(* IEC 61131-3 sources: AXOpen/src/components.abstractions/ctrl/src/AxoDrives (part 2) *)

(* ---- AxoDrive.st ---- *)
USING AXOpen.Core;
USING AXOpen.Messaging.Static;
USING AXOpen.Messaging;
USING System.Strings;

NAMESPACE AXOpen.Components.Abstractions.AxoDrives
    {#ix-attr:[Container(Layout.Wrap)]}
    CLASS PUBLIC ABSTRACT AxoDrive EXTENDS AXOpen.Core.AxoComponent IMPLEMENTS AXOpen.Components.Abstractions.AxoDrives.IAxoDrive
        VAR PUBLIC
            {#ix-attr:[Container(Layout.Wrap)]}
            {#ix-attr:[ComponentHeader()]}
            {#ix-attr:[ReadOnly()]}
            {#ix-set:AttributeName = "<#Drive state#>"}
            DriveState          :   AXOpen.Components.Abstractions.AxoDrives.eAxoDriveState;

            DriveStatus         :   AxoDrive_Status;
            Messenger           :   AXOpen.Messaging.Static.AxoMessenger;
            TaskMessenger       :   AXOpen.Messaging.Static.AxoMessenger;
        END_VAR

        VAR PUBLIC
            {#ix-attr:[Container(Layout.Wrap)]}
            {#ix-attr:[ComponentDetails("Tasks")]}
            {#ix-set:AttributeName = "<#Restore#>"}
            RestoreTask : AXOpen.Core.AxoTask;
            //***********Power********************************
            {#ix-attr:[Container(Layout.UniformGrid)]}
            {#ix-attr:[Group(GroupLayout.GroupBox)]}
            {#ix-attr:[ComponentDetails("Tasks")]}
            {#ix-set:AttributeName = "<#Power task#>"}
            AxoPower_Task                           :   AXOpen.Components.Abstractions.AxoDrives.Axo_Power;
            {#ix-attr:[ComponentDetails("Tasks")]}
            {#ix-set:AttributeName = "<#Power status#>"}
            AxoPower_Status                         :   BOOL;
            {#ix-attr:[ComponentDetails("Tasks")]}
            {#ix-set:AttributeName = "<#Power valid#>"}
            AxoPower_Valid                          :   BOOL;
            {#ix-attr:[ComponentDetails("Tasks")]}
            {#ix-set:AttributeName = "<#Power error#>"}
            AxoPower_Error                          :   BOOL;
            {#ix-attr:[ComponentDetails("Tasks")]}
            {#ix-set:AttributeName = "<#Power error ID#>"}
            AxoPower_ErrorID                        :   WORD;
            //***********Stop*********************************
            {#ix-attr:[Container(Layout.UniformGrid)]}
            {#ix-attr:[Group(GroupLayout.GroupBox)]}
            {#ix-attr:[ComponentDetails("Tasks")]}
            {#ix-set:AttributeName = "<#Stop task#>"}
            AxoStop_Task                            :   AXOpen.Core.AxoTask;
            {#ix-attr:[ComponentDetails("Tasks")]}
            {#ix-set:AttributeName = "<#Stop decceleration#>"}
            AxoStop_Deceleration                    :   LREAL;
            {#ix-attr:[ComponentDetails("Tasks")]}
            {#ix-set:AttributeName = "<#Stop jerk#>"}
            AxoStop_Jerk                            :   LREAL;
            {#ix-attr:[ComponentDetails("Tasks")]}
            {#ix-set:AttributeName = "<#Stop done#>"}
            AxoStop_Done                            :   BOOL;
            {#ix-attr:[ComponentDetails("Tasks")]}
            {#ix-set:AttributeName = "<#Stop busy#>"}
            AxoStop_Busy                            :   BOOL;
            {#ix-attr:[ComponentDetails("Tasks")]}
            {#ix-set:AttributeName = "<#Stop active#>"}
            AxoStop_Active                          :   BOOL;
            {#ix-attr:[ComponentDetails("Tasks")]}
            {#ix-set:AttributeName = "<#Stop aborted#>"}
            AxoStop_CommandAborted                  :   BOOL;
            {#ix-attr:[ComponentDetails("Tasks")]}
            {#ix-set:AttributeName = "<#Stop error#>"}
            AxoStop_Error                           :   BOOL;
            {#ix-attr:[ComponentDetails("Tasks")]}
            {#ix-set:AttributeName = "<#Stop error ID#>"}
            AxoStop_ErrorID                         :   WORD;
            //***********Halt*********************************
            {#ix-attr:[Container(Layout.UniformGrid)]}
            {#ix-attr:[Group(GroupLayout.GroupBox)]}
            {#ix-attr:[ComponentDetails("Tasks")]}
            {#ix-set:AttributeName = "<#Halt task#>"}
            AxoHalt_Task                            :   AXOpen.Core.AxoTask;
            {#ix-attr:[ComponentDetails("Tasks")]}
            {#ix-set:AttributeName = "<#Halt decceleration#>"}
            AxoHalt_Deceleration                    :   LREAL;
            {#ix-attr:[ComponentDetails("Tasks")]}
            {#ix-set:AttributeName = "<#Halt decceleration#>"}
            AxoHalt_Jerk                            :   LREAL;
            {#ix-attr:[ComponentDetails("Tasks")]}
            {#ix-set:AttributeName = "<#Halt done#>"}
            AxoHalt_Done                            :   BOOL;
            {#ix-attr:[ComponentDetails("Tasks")]}
            {#ix-set:AttributeName = "<#Halt busy#>"}
            AxoHalt_Busy                            :   BOOL;
            {#ix-attr:[ComponentDetails("Tasks")]}
            {#ix-set:AttributeName = "<#Halt active#>"}
            AxoHalt_Active                          :   BOOL;
            {#ix-attr:[ComponentDetails("Tasks")]}
            {#ix-set:AttributeName = "<#Halt aborted#>"}
            AxoHalt_CommandAborted                  :   BOOL;
            {#ix-attr:[ComponentDetails("Tasks")]}
            {#ix-set:AttributeName = "<#Halt error#>"}
            AxoHalt_Error                           :   BOOL;
            {#ix-attr:[ComponentDetails("Tasks")]}
            {#ix-set:AttributeName = "<#Halt error ID#>"}
            AxoHalt_ErrorID                         :   WORD;
            //***********Home*********************************
            {#ix-attr:[Container(Layout.UniformGrid)]}
            {#ix-attr:[Group(GroupLayout.GroupBox)]}
            {#ix-attr:[ComponentDetails("Tasks")]}
            {#ix-set:AttributeName = "<#Homming task#>"}
            AxoHome_Task                            :   AXOpen.Core.AxoTask;
            {#ix-attr:[ComponentDetails("Tasks")]}
            {#ix-set:AttributeName = "<#Homming position#>"}
            AxoHome_Position                        :   LREAL;
            {#ix-attr:[ComponentDetails("Tasks")]}
            {#ix-set:AttributeName = "<#Homming mode#>"}
            AxoHome_HommingMode                     :   INT;
            {#ix-attr:[ComponentDetails("Tasks")]}
            {#ix-set:AttributeName = "<#Homming velocity#>"}
            AxoHome_Velocity                        :   LREAL;
            {#ix-attr:[ComponentDetails("Tasks")]}
            {#ix-set:AttributeName = "<#Homming acceleration#>"}
            AxoHome_Acceleration                    :   LREAL;
            {#ix-attr:[ComponentDetails("Tasks")]}
            {#ix-set:AttributeName = "<#Homming decceleration#>"}
            AxoHome_Deceleration                    :   LREAL;
            {#ix-attr:[ComponentDetails("Tasks")]}
            {#ix-set:AttributeName = "<#Home status#>"}
            AxoHome_Status                          :   BOOL;
            {#ix-attr:[ComponentDetails("Tasks")]}
            {#ix-set:AttributeName = "<#Home valid#>"}
            AxoHome_Valid                           :   BOOL;
            {#ix-attr:[ComponentDetails("Tasks")]}
            {#ix-set:AttributeName = "<#Home error#>"}
            AxoHome_Error                           :   BOOL;
            {#ix-attr:[ComponentDetails("Tasks")]}
            {#ix-set:AttributeName = "<#Home error ID#>"}
            AxoHome_ErrorID                         :   WORD;
            {#ix-attr:[ComponentDetails("Tasks")]}
            {#ix-set:AttributeName = "<#Home done#>"}
            AxoHome_Done                            :   BOOL;
            {#ix-attr:[ComponentDetails("Tasks")]}
            {#ix-set:AttributeName = "<#Home busy#>"}
            AxoHome_Busy                            :   BOOL;
            {#ix-attr:[ComponentDetails("Tasks")]}
            {#ix-set:AttributeName = "<#Home active#>"}
            AxoHome_Active                          :   BOOL;
            {#ix-attr:[ComponentDetails("Tasks")]}
            {#ix-set:AttributeName = "<#Home aborted#>"}
            AxoHome_CommandAborted                  :   BOOL;
            //***********MoveAbsolute*************************
            {#ix-attr:[Container(Layout.UniformGrid)]}
            {#ix-attr:[Group(GroupLayout.GroupBox)]}
            {#ix-attr:[ComponentDetails("Tasks")]}
            {#ix-set:AttributeName = "<#Move absolute task#>"}
            AxoMoveAbsolute_Task                    :   AXOpen.Core.AxoTask;
            {#ix-attr:[ComponentDetails("Tasks")]}
            {#ix-set:AttributeName = "<#Move absolute continous update#>"}
            AxoMoveAbsolute_ContinuousUpdate        :   BOOL;
            {#ix-attr:[ComponentDetails("Tasks")]}
            {#ix-set:AttributeName = "<#Move absolute position#>"}
            AxoMoveAbsolute_Position                :   LREAL;
            {#ix-attr:[ComponentDetails("Tasks")]}
            {#ix-set:AttributeName = "<#Move absolute velocity#>"}
            AxoMoveAbsolute_Velocity                :   LREAL;
            {#ix-attr:[ComponentDetails("Tasks")]}
            {#ix-set:AttributeName = "<#Move absolute acceleration#>"}
            AxoMoveAbsolute_Acceleration            :   LREAL;
            {#ix-attr:[ComponentDetails("Tasks")]}
            {#ix-set:AttributeName = "<#Move absolute decceleration#>"}
            AxoMoveAbsolute_Deceleration            :   LREAL;
            {#ix-attr:[ComponentDetails("Tasks")]}
            {#ix-set:AttributeName = "<#Move absolute jerk#>"}
            AxoMoveAbsolute_Jerk                    :   LREAL;
            {#ix-attr:[ComponentDetails("Tasks")]}
            {#ix-set:AttributeName = "<#Move absolute direction#>"}
            AxoMoveAbsolute_Direction               :   AXOpen.Components.Abstractions.AxoDrives.eAxoDriveDirection;
            {#ix-attr:[ComponentDetails("Tasks")]}
            {#ix-set:AttributeName = "<#Move absolute done#>"}
            AxoMoveAbsolute_Done                    :   BOOL;
            {#ix-attr:[ComponentDetails("Tasks")]}
            {#ix-set:AttributeName = "<#Move absolute busy#>"}
            AxoMoveAbsolute_Busy                    :   BOOL;
            {#ix-attr:[ComponentDetails("Tasks")]}
            {#ix-set:AttributeName = "<#Move absolute active#>"}
            AxoMoveAbsolute_Active                  :   BOOL;
            {#ix-attr:[ComponentDetails("Tasks")]}
            {#ix-set:AttributeName = "<#Move absolute aborted#>"}
            AxoMoveAbsolute_CommandAborted          :   BOOL;
            {#ix-attr:[ComponentDetails("Tasks")]}
            {#ix-set:AttributeName = "<#Move absolute error#>"}
            AxoMoveAbsolute_Error                   :   BOOL;
            {#ix-attr:[ComponentDetails("Tasks")]}
            {#ix-set:AttributeName = "<#Move absolute error ID#>"}
            AxoMoveAbsolute_ErrorID                 :   WORD;
            //***********MoveRelative*************************
            {#ix-attr:[Container(Layout.UniformGrid)]}
            {#ix-attr:[Group(GroupLayout.GroupBox)]}
            {#ix-attr:[ComponentDetails("Tasks")]}
            {#ix-set:AttributeName = "<#Move relative task#>"}
            AxoMoveRelative_Task                    :   AXOpen.Core.AxoTask;
            {#ix-attr:[ComponentDetails("Tasks")]}
            {#ix-set:AttributeName = "<#Move relative continuous update#>"}
            AxoMoveRelative_ContinuousUpdate        :   BOOL;
            {#ix-attr:[ComponentDetails("Tasks")]}
            {#ix-set:AttributeName = "<#Move relative distance#>"}
            AxoMoveRelative_Distance                :   LREAL;
            {#ix-attr:[ComponentDetails("Tasks")]}
            {#ix-set:AttributeName = "<#Move relative velocity#>"}
            AxoMoveRelative_Velocity                :   LREAL;
            {#ix-attr:[ComponentDetails("Tasks")]}
            {#ix-set:AttributeName = "<#Move relative acceleration#>"}
            AxoMoveRelative_Acceleration            :   LREAL;
            {#ix-attr:[ComponentDetails("Tasks")]}
            {#ix-set:AttributeName = "<#Move relative deceleration#>"}
            AxoMoveRelative_Deceleration            :   LREAL;
            {#ix-attr:[ComponentDetails("Tasks")]}
            {#ix-set:AttributeName = "<#Move relative jerk#>"}
            AxoMoveRelative_Jerk                    :   LREAL;
            {#ix-attr:[ComponentDetails("Tasks")]}
            {#ix-set:AttributeName = "<#Move relative direction#>"}
            AxoMoveRelative_Direction               :   AXOpen.Components.Abstractions.AxoDrives.eAxoDriveDirection;
            {#ix-attr:[ComponentDetails("Tasks")]}
            {#ix-set:AttributeName = "<#Move relative done#>"}
            AxoMoveRelative_Done                    :   BOOL;
            {#ix-attr:[ComponentDetails("Tasks")]}
            {#ix-set:AttributeName = "<#Move relative busy#>"}
            AxoMoveRelative_Busy                    :   BOOL;
            {#ix-attr:[ComponentDetails("Tasks")]}
            {#ix-set:AttributeName = "<#Move relative active#>"}
            AxoMoveRelative_Active                  :   BOOL;
            {#ix-attr:[ComponentDetails("Tasks")]}
            {#ix-set:AttributeName = "<#Move relative aborted#>"}
            AxoMoveRelative_CommandAborted          :   BOOL;
            {#ix-attr:[ComponentDetails("Tasks")]}
            {#ix-set:AttributeName = "<#Move relative error#>"}
            AxoMoveRelative_Error                   :   BOOL;
            {#ix-attr:[ComponentDetails("Tasks")]}
            {#ix-set:AttributeName = "<#Move relative error ID#>"}
            AxoMoveRelative_ErrorID                 :   WORD;
            //***********MoveAdditive*************************
            {#ix-attr:[Container(Layout.UniformGrid)]}
            {#ix-attr:[Group(GroupLayout.GroupBox)]}
            {#ix-attr:[ComponentDetails("Tasks")]}
            {#ix-set:AttributeName = "<#Move additive task#>"}
            AxoMoveAdditive_Task                    :   AXOpen.Core.AxoTask;
            {#ix-attr:[ComponentDetails("Tasks")]}
            {#ix-set:AttributeName = "<#Move additive continuous update#>"}
            AxoMoveAdditive_ContinuousUpdate        :   BOOL;
            {#ix-attr:[ComponentDetails("Tasks")]}
            {#ix-set:AttributeName = "<#Move additive distance#>"}
            AxoMoveAdditive_Distance                :   LREAL;
            {#ix-attr:[ComponentDetails("Tasks")]}
            {#ix-set:AttributeName = "<#Move additive velocity#>"}
            AxoMoveAdditive_Velocity                :   LREAL;
            {#ix-attr:[ComponentDetails("Tasks")]}
            {#ix-set:AttributeName = "<#Move additive acceleration#>"}
            AxoMoveAdditive_Acceleration            :   LREAL;
            {#ix-attr:[ComponentDetails("Tasks")]}
            {#ix-set:AttributeName = "<#Move additive deceleration#>"}
            AxoMoveAdditive_Deceleration            :   LREAL;
            {#ix-attr:[ComponentDetails("Tasks")]}
            {#ix-set:AttributeName = "<#Move additive jerk#>"}
            AxoMoveAdditive_Jerk                    :   LREAL;
            {#ix-attr:[ComponentDetails("Tasks")]}
            {#ix-set:AttributeName = "<#Move additive direction#>"}
            AxoMoveAdditive_Direction               :   AXOpen.Components.Abstractions.AxoDrives.eAxoDriveDirection;
            {#ix-attr:[ComponentDetails("Tasks")]}
            {#ix-set:AttributeName = "<#Move additive done#>"}
            AxoMoveAdditive_Done                    :   BOOL;
            {#ix-attr:[ComponentDetails("Tasks")]}
            {#ix-set:AttributeName = "<#Move additive busy#>"}
            AxoMoveAdditive_Busy                    :   BOOL;
            {#ix-attr:[ComponentDetails("Tasks")]}
            {#ix-set:AttributeName = "<#Move additive active#>"}
            AxoMoveAdditive_Active                  :   BOOL;
            {#ix-attr:[ComponentDetails("Tasks")]}
            {#ix-set:AttributeName = "<#Move additive aborted#>"}
            AxoMoveAdditive_CommandAborted          :   BOOL;
            {#ix-attr:[ComponentDetails("Tasks")]}
            {#ix-set:AttributeName = "<#Move additive error#>"}
            AxoMoveAdditive_Error                   :   BOOL;
            {#ix-attr:[ComponentDetails("Tasks")]}
            {#ix-set:AttributeName = "<#Move additive error ID#>"}
            AxoMoveAdditive_ErrorID                 :   WORD;
            //***********MoveVelocity*************************
            {#ix-attr:[Container(Layout.UniformGrid)]}
            {#ix-attr:[Group(GroupLayout.GroupBox)]}
            {#ix-attr:[ComponentDetails("Tasks")]}
            {#ix-set:AttributeName = "<#Move velocity task#>"}
            AxoMoveVelocity_Task                    :   AXOpen.Core.AxoTask;
            {#ix-attr:[ComponentDetails("Tasks")]}
            {#ix-set:AttributeName = "<#Move velocity continuous update#>"}
            AxoMoveVelocity_ContinuousUpdate        :   BOOL;
            {#ix-attr:[ComponentDetails("Tasks")]}
            {#ix-set:AttributeName = "<#Move velocity velocity#>"}
            AxoMoveVelocity_Velocity                :   LREAL;
            {#ix-attr:[ComponentDetails("Tasks")]}
            {#ix-set:AttributeName = "<#Move velocity acceleration#>"}
            AxoMoveVelocity_Acceleration            :   LREAL;
            {#ix-attr:[ComponentDetails("Tasks")]}
            {#ix-set:AttributeName = "<#Move velocity deceleration#>"}
            AxoMoveVelocity_Deceleration            :   LREAL;
            {#ix-attr:[ComponentDetails("Tasks")]}
            {#ix-set:AttributeName = "<#Move velocity jerk#>"}
            AxoMoveVelocity_Jerk                    :   LREAL;
            {#ix-attr:[ComponentDetails("Tasks")]}
            {#ix-set:AttributeName = "<#Move velocity #>"}
            AxoMoveVelocity_Direction               :   AXOpen.Components.Abstractions.AxoDrives.eAxoDriveDirection;
            {#ix-attr:[ComponentDetails("Tasks")]}
            {#ix-set:AttributeName = "<#Move velocity in velocity#>"}
            AxoMoveVelocity_InVelocity              :   BOOL;
            {#ix-attr:[ComponentDetails("Tasks")]}
            {#ix-set:AttributeName = "<#Move velocity busy#>"}
            AxoMoveVelocity_Busy                    :   BOOL;
            {#ix-attr:[ComponentDetails("Tasks")]}
            {#ix-set:AttributeName = "<#Move velocity active#>"}
            AxoMoveVelocity_Active                  :   BOOL;
            {#ix-attr:[ComponentDetails("Tasks")]}
            {#ix-set:AttributeName = "<#Move velocity aborted#>"}
            AxoMoveVelocity_CommandAborted          :   BOOL;
            {#ix-attr:[ComponentDetails("Tasks")]}
            {#ix-set:AttributeName = "<#Move velocity error#>"}
            AxoMoveVelocity_Error                   :   BOOL;
            {#ix-attr:[ComponentDetails("Tasks")]}
            {#ix-set:AttributeName = "<#Move velocity error ID#>"}
            AxoMoveVelocity_ErrorID                 :   WORD;

            //***********TorqueControl************************
            {#ix-attr:[Container(Layout.UniformGrid)]}
            {#ix-attr:[Group(GroupLayout.GroupBox)]}
            {#ix-attr:[ComponentDetails("Tasks")]}
            {#ix-set:AttributeName = "<#Move torque task#>"}
            AxoTorqueControl_Task                   :   AXOpen.Core.AxoTask;
            {#ix-attr:[ComponentDetails("Tasks")]}
            {#ix-set:AttributeName = "<#Move torque continuous update#>"}
            AxoTorqueControl_ContinuousUpdate       :   BOOL;
            {#ix-attr:[ComponentDetails("Tasks")]}
            {#ix-set:AttributeName = "<#Move torque torque#>"}
            AxoTorqueControl_Torque                 :   LREAL;
            {#ix-attr:[ComponentDetails("Tasks")]}
            {#ix-set:AttributeName = "<#Move torque torque ramp#>"}
            AxoTorqueControl_TorqueRamp             :   LREAL;
            {#ix-attr:[ComponentDetails("Tasks")]}
            {#ix-set:AttributeName = "<#Move torque velocity#>"}
            AxoTorqueControl_Velocity               :   LREAL;
            {#ix-attr:[ComponentDetails("Tasks")]}
            {#ix-set:AttributeName = "<#Move torque acceleration#>"}
            AxoTorqueControl_Acceleration           :   LREAL;
            {#ix-attr:[ComponentDetails("Tasks")]}
            {#ix-set:AttributeName = "<#Move torque deceleration#>"}
            AxoTorqueControl_Deceleration           :   LREAL;
            {#ix-attr:[ComponentDetails("Tasks")]}
            {#ix-set:AttributeName = "<#Move torque jerk#>"}
            AxoTorqueControl_Jerk                   :   LREAL;
            {#ix-attr:[ComponentDetails("Tasks")]}
            {#ix-set:AttributeName = "<#Move torque direction#>"}
            AxoTorqueControl_Direction              :   AXOpen.Components.Abstractions.AxoDrives.eAxoDriveDirection;
            {#ix-attr:[ComponentDetails("Tasks")]}
            {#ix-set:AttributeName = "<#Move torque in torque#>"}
            AxoTorqueControl_InTorque               :   BOOL;
            {#ix-attr:[ComponentDetails("Tasks")]}
            {#ix-set:AttributeName = "<#Move torque busy#>"}
            AxoTorqueControl_Busy                   :   BOOL;
            {#ix-attr:[ComponentDetails("Tasks")]}
            {#ix-set:AttributeName = "<#Move torque active#>"}
            AxoTorqueControl_Active                 :   BOOL;
            {#ix-attr:[ComponentDetails("Tasks")]}
            {#ix-set:AttributeName = "<#Move torque aborted#>"}
            AxoTorqueControl_CommandAborted         :   BOOL;
            {#ix-attr:[ComponentDetails("Tasks")]}
            {#ix-set:AttributeName = "<#Move torque error#>"}
            AxoTorqueControl_Error                  :   BOOL;
            {#ix-attr:[ComponentDetails("Tasks")]}
            {#ix-set:AttributeName = "<#Move torque error ID#>"}
            AxoTorqueControl_ErrorID                :   WORD;
            //***********SetPosition**************************
            {#ix-attr:[Container(Layout.UniformGrid)]}
            {#ix-attr:[Group(GroupLayout.GroupBox)]}
            {#ix-attr:[ComponentDetails("Tasks")]}
            {#ix-set:AttributeName = "<#Set position task#>"}
            AxoSetPosition_Task                     :   AXOpen.Core.AxoTask;
            {#ix-attr:[ComponentDetails("Tasks")]}
            {#ix-set:AttributeName = "<#Set position position#>"}
            AxoSetPosition_Position                 :   REAL;
            {#ix-attr:[ComponentDetails("Tasks")]}
            {#ix-set:AttributeName = "<#Set position relative#>"}
            AxoSetPosition_Relative                 :   BOOL;
            {#ix-attr:[ComponentDetails("Tasks")]}
            {#ix-set:AttributeName = "<#Set position execution mode#>"}
            AxoSetPosition_ExecutionMode            :   AXOpen.Components.Abstractions.AxoDrives.eAxoExecutionMode;
            {#ix-attr:[ComponentDetails("Tasks")]}
            {#ix-set:AttributeName = "<#Set position done#>"}
            AxoSetPosition_Done                     :   BOOL;
            {#ix-attr:[ComponentDetails("Tasks")]}
            {#ix-set:AttributeName = "<#Set position error#>"}
            AxoSetPosition_Error                    :   BOOL;
            {#ix-attr:[ComponentDetails("Tasks")]}
            {#ix-set:AttributeName = "<#Set position error ID#>"}
            AxoSetPosition_ErrorID                  :   WORD;
            //***********SetOverride**************************
            {#ix-attr:[Container(Layout.UniformGrid)]}
            {#ix-attr:[Group(GroupLayout.GroupBox)]}
            {#ix-attr:[ComponentDetails("Tasks")]}
            {#ix-set:AttributeName = "<#Set override task#>"}
            AxoSetOverride_Task                     :   AXOpen.Core.AxoToggleTask;
            {#ix-attr:[ComponentDetails("Tasks")]}
            {#ix-set:AttributeName = "<#Set override velocity factor#>"}
            AxoSetOverride_VelFactor                :   LREAL;
            {#ix-attr:[ComponentDetails("Tasks")]}
            {#ix-set:AttributeName = "<#Set override acceleration factor#>"}
            AxoSetOverride_AccFactor                :   LREAL;
            {#ix-attr:[ComponentDetails("Tasks")]}
            {#ix-set:AttributeName = "<#Set override jerk factor#>"}
            AxoSetOverride_JerkFactor               :   LREAL;
            {#ix-attr:[ComponentDetails("Tasks")]}
            {#ix-set:AttributeName = "<#Set override enabled#>"}
            AxoSetOverride_Enabled                  :   BOOL;
            {#ix-attr:[ComponentDetails("Tasks")]}
            {#ix-set:AttributeName = "<#Set override busy#>"}
            AxoSetOverride_Busy                     :   BOOL;
            {#ix-attr:[ComponentDetails("Tasks")]}
            {#ix-set:AttributeName = "<#Set override error#>"}
            AxoSetOverride_Error                    :   BOOL;
            {#ix-attr:[ComponentDetails("Tasks")]}
            {#ix-set:AttributeName = "<#Set override error ID#>"}
            AxoSetOverride_ErrorID                  :   WORD;
            //***********ReadParameter************************
            {#ix-attr:[Container(Layout.UniformGrid)]}
            {#ix-attr:[Group(GroupLayout.GroupBox)]}
            {#ix-attr:[ComponentDetails("Tasks")]}
            {#ix-set:AttributeName = "<#Read parameter task#>"}
            AxoReadParameter_Task                   :   AXOpen.Core.AxoToggleTask;
            {#ix-attr:[ComponentDetails("Tasks")]}
            {#ix-set:AttributeName = "<#Read parameter number#>"}
            AxoReadParameter_ParameterNumber        :   INT;
            {#ix-attr:[ComponentDetails("Tasks")]}
            {#ix-set:AttributeName = "<#Read parameter valid#>"}
            AxoReadParameter_Valid                  :   BOOL;
            {#ix-attr:[ComponentDetails("Tasks")]}
            {#ix-set:AttributeName = "<#Read parameter busy#>"}
            AxoReadParameter_Busy                   :   BOOL;
            {#ix-attr:[ComponentDetails("Tasks")]}
            {#ix-set:AttributeName = "<#Read parameter error#>"}
            AxoReadParameter_Error                  :   BOOL;
            {#ix-attr:[ComponentDetails("Tasks")]}
            {#ix-set:AttributeName = "<#Read parameter error ID#>"}
            AxoReadParameter_ErrorID                :   WORD;
            {#ix-attr:[ComponentDetails("Tasks")]}
            {#ix-set:AttributeName = "<#Read parameter value#>"}
            AxoReadParameter_Value                  :   REAL;
            //***********ReadBoolParameter********************
            {#ix-attr:[Container(Layout.UniformGrid)]}
            {#ix-attr:[Group(GroupLayout.GroupBox)]}
            {#ix-attr:[ComponentDetails("Tasks")]}
            {#ix-set:AttributeName = "<#Read bool parameter task#>"}
            AxoReadBoolParameter_Task               :   AXOpen.Core.AxoToggleTask;
            {#ix-attr:[ComponentDetails("Tasks")]}
            {#ix-set:AttributeName = "<#Read bool parameter number#>"}
            AxoReadBoolParameter_ParameterNumber    :   INT;
            {#ix-attr:[ComponentDetails("Tasks")]}
            {#ix-set:AttributeName = "<#Read bool parameter valid#>"}
            AxoReadBoolParameter_Valid              :   BOOL;
            {#ix-attr:[ComponentDetails("Tasks")]}
            {#ix-set:AttributeName = "<#Read bool parameter busy#>"}
            AxoReadBoolParameter_Busy               :   BOOL;
            {#ix-attr:[ComponentDetails("Tasks")]}
            {#ix-set:AttributeName = "<#Read bool parameter error#>"}
            AxoReadBoolParameter_Error              :   BOOL;
            {#ix-attr:[ComponentDetails("Tasks")]}
            {#ix-set:AttributeName = "<#Read bool parameter error ID#>"}
            AxoReadBoolParameter_ErrorID            :   WORD;
            {#ix-attr:[ComponentDetails("Tasks")]}
            {#ix-set:AttributeName = "<#Read bool parameter value#>"}
            AxoReadBoolParameter_Value              :   BOOL;
            //***********WriteParameter***********************
            {#ix-attr:[Container(Layout.UniformGrid)]}
            {#ix-attr:[Group(GroupLayout.GroupBox)]}
            {#ix-attr:[ComponentDetails("Tasks")]}
            {#ix-set:AttributeName = "<#Write parameter task#>"}
            AxoWriteParameter_Task                  :   AXOpen.Core.AxoTask;
            {#ix-attr:[ComponentDetails("Tasks")]}
            {#ix-set:AttributeName = "<#Write parameter number#>"}
            AxoWriteParameter_ParameterNumber       :   INT;
            {#ix-attr:[ComponentDetails("Tasks")]}
            {#ix-set:AttributeName = "<#Write parameter value#>"}
            AxoWriteParameter_Value                 :   REAL;
            {#ix-attr:[ComponentDetails("Tasks")]}
            {#ix-set:AttributeName = "<#Write parameter execution mode#>"}
            AxoWriteParameter_ExecutionMode         :   AXOpen.Components.Abstractions.AxoDrives.eAxoExecutionMode;
            {#ix-attr:[ComponentDetails("Tasks")]}
            {#ix-set:AttributeName = "<#Write parameter done#>"}
            AxoWriteParameter_Done                  :   BOOL;
            {#ix-attr:[ComponentDetails("Tasks")]}
            {#ix-set:AttributeName = "<#Write parameter busy#>"}
            AxoWriteParameter_Busy                  :   BOOL;
            {#ix-attr:[ComponentDetails("Tasks")]}
            {#ix-set:AttributeName = "<#Write parameter error#>"}
            AxoWriteParameter_Error                 :   BOOL;
            {#ix-attr:[ComponentDetails("Tasks")]}
            {#ix-set:AttributeName = "<#Write parameter error ID#>"}
            AxoWriteParameter_ErrorID               :   WORD;
            //***********WriteBoolParameter*******************
            {#ix-attr:[Container(Layout.UniformGrid)]}
            {#ix-attr:[Group(GroupLayout.GroupBox)]}
            {#ix-attr:[ComponentDetails("Tasks")]}
            {#ix-set:AttributeName = "<#Write bool parameter task#>"}
            AxoWriteBoolParameter_Task              :   AXOpen.Core.AxoTask;
            {#ix-attr:[ComponentDetails("Tasks")]}
            {#ix-set:AttributeName = "<#Write bool parameter number#>"}
            AxoWriteBoolParameter_ParameterNumber   :   INT;
            {#ix-attr:[ComponentDetails("Tasks")]}
            {#ix-set:AttributeName = "<#Write bool parameter value#>"}
            AxoWriteBoolParameter_Value             :   BOOL;
            {#ix-attr:[ComponentDetails("Tasks")]}
            {#ix-set:AttributeName = "<#Write bool parameter execution mode#>"}
            AxoWriteBoolParameter_ExecutionMode     :   AXOpen.Components.Abstractions.AxoDrives.eAxoExecutionMode;
            {#ix-attr:[ComponentDetails("Tasks")]}
            {#ix-set:AttributeName = "<#Write bool parameter done#>"}
            AxoWriteBoolParameter_Done              :   BOOL;
            {#ix-attr:[ComponentDetails("Tasks")]}
            {#ix-set:AttributeName = "<#Write bool parameter busy#>"}
            AxoWriteBoolParameter_Busy              :   BOOL;
            {#ix-attr:[ComponentDetails("Tasks")]}
            {#ix-set:AttributeName = "<#Write bool parameter error#>"}
            AxoWriteBoolParameter_Error             :   BOOL;
            {#ix-attr:[ComponentDetails("Tasks")]}
            {#ix-set:AttributeName = "<#Write bool parameter error ID#>"}
            AxoWriteBoolParameter_ErrorID           :   WORD;
            //***********ReadDigitalInput*********************
            {#ix-attr:[Container(Layout.UniformGrid)]}
            {#ix-attr:[Group(GroupLayout.GroupBox)]}
            {#ix-attr:[ComponentDetails("Tasks")]}
            {#ix-set:AttributeName = "<#Read digital input task#>"}
            AxoReadDigitalInput_Task                :   AXOpen.Core.AxoToggleTask;
            {#ix-attr:[ComponentDetails("Tasks")]}
            {#ix-set:AttributeName = "<#Read digital input number#>"}
            AxoReadDigitalInput_InputNumber         :   INT;
            {#ix-attr:[ComponentDetails("Tasks")]}
            {#ix-set:AttributeName = "<#Read digital input valid#>"}
            AxoReadDigitalInput_Valid               :   BOOL;
            {#ix-attr:[ComponentDetails("Tasks")]}
            {#ix-set:AttributeName = "<#Read digital input busy#>"}
            AxoReadDigitalInput_Busy                :   BOOL;
            {#ix-attr:[ComponentDetails("Tasks")]}
            {#ix-set:AttributeName = "<#Read digital input error#>"}
            AxoReadDigitalInput_Error               :   BOOL;
            {#ix-attr:[ComponentDetails("Tasks")]}
            {#ix-set:AttributeName = "<#Read digital input error ID#>"}
            AxoReadDigitalInput_ErrorID             :   WORD;
            {#ix-attr:[ComponentDetails("Tasks")]}
            {#ix-set:AttributeName = "<#Read digital input value#>"}
            AxoReadDigitalInput_Value               :   BOOL;
            //***********ReadDigitalOutput********************
            {#ix-attr:[Container(Layout.UniformGrid)]}
            {#ix-attr:[Group(GroupLayout.GroupBox)]}
            {#ix-attr:[ComponentDetails("Tasks")]}
            {#ix-set:AttributeName = "<#Read digital output task#>"}
            AxoReadDigitalOutput_Task               :   AXOpen.Core.AxoToggleTask;
            {#ix-attr:[ComponentDetails("Tasks")]}
            {#ix-set:AttributeName = "<#Read digital output number#>"}
            AxoReadDigitalOutput_OutputNumber       :   INT;
            {#ix-attr:[ComponentDetails("Tasks")]}
            {#ix-set:AttributeName = "<#Read digital output valid#>"}
            AxoReadDigitalOutput_Valid              :   BOOL;
            {#ix-attr:[ComponentDetails("Tasks")]}
            {#ix-set:AttributeName = "<#Read digital output busy#>"}
            AxoReadDigitalOutput_Busy               :   BOOL;
            {#ix-attr:[ComponentDetails("Tasks")]}
            {#ix-set:AttributeName = "<#Read digital output error#>"}
            AxoReadDigitalOutput_Error              :   BOOL;
            {#ix-attr:[ComponentDetails("Tasks")]}
            {#ix-set:AttributeName = "<#Read digital output error ID#>"}
            AxoReadDigitalOutput_ErrorID            :   WORD;
            {#ix-attr:[ComponentDetails("Tasks")]}
            {#ix-set:AttributeName = "<#Read digital output value#>"}
            AxoReadDigitalOutput_Value              :   BOOL;
            //***********WriteDigitalOutput*******************
            {#ix-attr:[Container(Layout.UniformGrid)]}
            {#ix-attr:[Group(GroupLayout.GroupBox)]}
            {#ix-attr:[ComponentDetails("Tasks")]}
            {#ix-set:AttributeName = "<#Write digital output task#>"}
            AxoWriteDigitalOutput_Task              :   AXOpen.Core.AxoTask;
            {#ix-attr:[ComponentDetails("Tasks")]}
            {#ix-set:AttributeName = "<#Write digital output number#>"}
            AxoWriteDigitalOutput_OutputNumber      :   INT;
            {#ix-attr:[ComponentDetails("Tasks")]}
            {#ix-set:AttributeName = "<#Write digital output value#>"}
            AxoWriteDigitalOutput_Value             :   BOOL;
            {#ix-attr:[ComponentDetails("Tasks")]}
            {#ix-set:AttributeName = "<#Write digital output execution mode#>"}
            AxoWriteDigitalOutput_ExecutionMode     :   AXOpen.Components.Abstractions.AxoDrives.eAxoExecutionMode;
            {#ix-attr:[ComponentDetails("Tasks")]}
            {#ix-set:AttributeName = "<#Write digital output done#>"}
            AxoWriteDigitalOutput_Done              :   BOOL;
            {#ix-attr:[ComponentDetails("Tasks")]}
            {#ix-set:AttributeName = "<#Write digital output busy#>"}
            AxoWriteDigitalOutput_Busy              :   BOOL;
            {#ix-attr:[ComponentDetails("Tasks")]}
            {#ix-set:AttributeName = "<#Write digital output error#>"}
            AxoWriteDigitalOutput_Error             :   BOOL;
            {#ix-attr:[ComponentDetails("Tasks")]}
            {#ix-set:AttributeName = "<#Write digital output error ID#>"}
            AxoWriteDigitalOutput_ErrorID           :   WORD;
            //***********ReadActualPosition*******************
            {#ix-attr:[Container(Layout.UniformGrid)]}
            {#ix-attr:[Group(GroupLayout.GroupBox)]}
            {#ix-attr:[ComponentDetails("Tasks")]}
            {#ix-set:AttributeName = "<#Read actual position task#>"}
            AxoReadActualPosition_Task              :   AXOpen.Core.AxoToggleTask;
            {#ix-attr:[ComponentDetails("Tasks")]}
            {#ix-set:AttributeName = "<#Read actual position valid#>"}
            AxoReadActualPosition_Valid             :   BOOL;
            {#ix-attr:[ComponentDetails("Tasks")]}
            {#ix-set:AttributeName = "<#Read actual position busy#>"}
            AxoReadActualPosition_Busy              :   BOOL;
            {#ix-attr:[ComponentDetails("Tasks")]}
            {#ix-set:AttributeName = "<#Read actual position error#>"}
            AxoReadActualPosition_Error             :   BOOL;
            {#ix-attr:[ComponentDetails("Tasks")]}
            {#ix-set:AttributeName = "<#Read actual position error ID#>"}
            AxoReadActualPosition_ErrorID           :   WORD;
            {#ix-attr:[ComponentDetails("Tasks")]}
            {#ix-set:AttributeName = "<#Read actual position value#>"}
            AxoReadActualPosition_Value             :   REAL;
            //***********ReadActualVelocity*******************
            {#ix-attr:[Container(Layout.UniformGrid)]}
            {#ix-attr:[Group(GroupLayout.GroupBox)]}
            {#ix-attr:[ComponentDetails("Tasks")]}
            {#ix-set:AttributeName = "<#Read actual velocity task#>"}
            AxoReadActualVelocity_Task              :   AXOpen.Core.AxoToggleTask;
            {#ix-attr:[ComponentDetails("Tasks")]}
            {#ix-set:AttributeName = "<#Read actual velocity valid#>"}
            AxoReadActualVelocity_Valid             :   BOOL;
            {#ix-attr:[ComponentDetails("Tasks")]}
            {#ix-set:AttributeName = "<#Read actual velocity busy#>"}
            AxoReadActualVelocity_Busy              :   BOOL;
            {#ix-attr:[ComponentDetails("Tasks")]}
            {#ix-set:AttributeName = "<#Read actual velocity error#>"}
            AxoReadActualVelocity_Error             :   BOOL;
            {#ix-attr:[ComponentDetails("Tasks")]}
            {#ix-set:AttributeName = "<#Read actual velocity error ID#>"}
            AxoReadActualVelocity_ErrorID           :   WORD;
            {#ix-attr:[ComponentDetails("Tasks")]}
            {#ix-set:AttributeName = "<#Read actual velocity value#>"}
            AxoReadActualVelocity_Value             :   REAL;
            //***********ReadActualTorque*********************
            {#ix-attr:[Container(Layout.UniformGrid)]}
            {#ix-attr:[Group(GroupLayout.GroupBox)]}
            {#ix-attr:[ComponentDetails("Tasks")]}
            {#ix-set:AttributeName = "<#Read actual torque task#>"}
            AxoReadActualTorque_Task                :   AXOpen.Core.AxoToggleTask;
            {#ix-attr:[ComponentDetails("Tasks")]}
            {#ix-set:AttributeName = "<#Read actual torque valid#>"}
            AxoReadActualTorque_Valid               :   BOOL;
            {#ix-attr:[ComponentDetails("Tasks")]}
            {#ix-set:AttributeName = "<#Read actual torque busy#>"}
            AxoReadActualTorque_Busy                :   BOOL;
            {#ix-attr:[ComponentDetails("Tasks")]}
            {#ix-set:AttributeName = "<#Read actual torque error#>"}
            AxoReadActualTorque_Error               :   BOOL;
            {#ix-attr:[ComponentDetails("Tasks")]}
            {#ix-set:AttributeName = "<#Read actual torque error ID#>"}
            AxoReadActualTorque_ErrorID             :   WORD;
            {#ix-attr:[ComponentDetails("Tasks")]}
            {#ix-set:AttributeName = "<#Read actual torque value#>"}
            AxoReadActualTorque_Value               :   REAL;
            //***********ReadStatus***************************
            {#ix-attr:[Container(Layout.UniformGrid)]}
            {#ix-attr:[Group(GroupLayout.GroupBox)]}
            {#ix-attr:[ComponentDetails("Tasks")]}
            {#ix-set:AttributeName = "<#Read status task#>"}
            AxoReadStatus_Task                      :   AXOpen.Core.AxoToggleTask;
            {#ix-attr:[ComponentDetails("Tasks")]}
            {#ix-set:AttributeName = "<#Read status valid#>"}
            AxoReadStatus_Valid                     :   BOOL;
            {#ix-attr:[ComponentDetails("Tasks")]}
            {#ix-set:AttributeName = "<#Read status busy#>"}
            AxoReadStatus_Busy                      :   BOOL;
            {#ix-attr:[ComponentDetails("Tasks")]}
            {#ix-set:AttributeName = "<#Read status error#>"}
            AxoReadStatus_Error                     :   BOOL;
            {#ix-attr:[ComponentDetails("Tasks")]}
            {#ix-set:AttributeName = "<#Read status error ID#>"}
            AxoReadStatus_ErrorID                   :   WORD;
            {#ix-attr:[ComponentDetails("Tasks")]}
            {#ix-set:AttributeName = "<#Read status error stop#>"}
            AxoReadStatus_ErrorStop                 :   BOOL;
            {#ix-attr:[ComponentDetails("Tasks")]}
            {#ix-set:AttributeName = "<#Read status disabled#>"}
            AxoReadStatus_Disabled                  :   BOOL;
            {#ix-attr:[ComponentDetails("Tasks")]}
            {#ix-set:AttributeName = "<#Read status stopping#>"}
            AxoReadStatus_Stopping                  :   BOOL;
            {#ix-attr:[ComponentDetails("Tasks")]}
            {#ix-set:AttributeName = "<#Read status homming#>"}
            AxoReadStatus_Homing                    :   BOOL;
            {#ix-attr:[ComponentDetails("Tasks")]}
            {#ix-set:AttributeName = "<#Read status standstill#>"}
            AxoReadStatus_Standstill                :   BOOL;
            {#ix-attr:[ComponentDetails("Tasks")]}
            {#ix-set:AttributeName = "<#Read status discrete motion#>"}
            AxoReadStatus_DiscreteMotion            :   BOOL;
            {#ix-attr:[ComponentDetails("Tasks")]}
            {#ix-set:AttributeName = "<#Read status continuous motion#>"}
            AxoReadStatus_ContinuousMotion          :   BOOL;
            {#ix-attr:[ComponentDetails("Tasks")]}
            {#ix-set:AttributeName = "<#Read status synchronized motion#>"}
            AxoReadStatus_SynchronizedMotion        :   BOOL;
            //***********ReadMotionState**********************
            {#ix-attr:[Container(Layout.UniformGrid)]}
            {#ix-attr:[Group(GroupLayout.GroupBox)]}
            {#ix-attr:[ComponentDetails("Tasks")]}
            {#ix-set:AttributeName = "<#Read motion state task#>"}
            AxoReadMotionState_Task                 :   AXOpen.Core.AxoToggleTask;
            {#ix-attr:[ComponentDetails("Tasks")]}
            {#ix-set:AttributeName = "<#Read motion state source#>"}
            AxoReadMotionState_Source               :   AXOpen.Components.Abstractions.AxoDrives.eAxoSource;
            {#ix-attr:[ComponentDetails("Tasks")]}
            {#ix-set:AttributeName = "<#Read motion state valid#>"}
            AxoReadMotionState_Valid                :   BOOL;
            {#ix-attr:[ComponentDetails("Tasks")]}
            {#ix-set:AttributeName = "<#Read motion state busy#>"}
            AxoReadMotionState_Busy                 :   BOOL;
            {#ix-attr:[ComponentDetails("Tasks")]}
            {#ix-set:AttributeName = "<#Read motion state error#>"}
            AxoReadMotionState_Error                :   BOOL;
            {#ix-attr:[ComponentDetails("Tasks")]}
            {#ix-set:AttributeName = "<#Read motion state error ID#>"}
            AxoReadMotionState_ErrorID              :   WORD;
            {#ix-attr:[ComponentDetails("Tasks")]}
            {#ix-set:AttributeName = "<#Read motion state constant velocity#>"}
            AxoReadMotionState_ConstantVelocity     :   BOOL;
            {#ix-attr:[ComponentDetails("Tasks")]}
            {#ix-set:AttributeName = "<#Read motion state accelerating#>"}
            AxoReadMotionState_Accelerating         :   BOOL;
            {#ix-attr:[ComponentDetails("Tasks")]}
            {#ix-set:AttributeName = "<#Read motion state decelerating#>"}
            AxoReadMotionState_Decelerating         :   BOOL;
            {#ix-attr:[ComponentDetails("Tasks")]}
            {#ix-set:AttributeName = "<#Read motion state direction positive#>"}
            AxoReadMotionState_DirectionPositive    :   BOOL;
            {#ix-attr:[ComponentDetails("Tasks")]}
            {#ix-set:AttributeName = "<#Read motion state direction negative#>"}
            AxoReadMotionState_DirectionNegative    :   BOOL;
            //***********ReadAxisInfo*************************
            {#ix-attr:[Container(Layout.UniformGrid)]}
            {#ix-attr:[Group(GroupLayout.GroupBox)]}
            {#ix-attr:[ComponentDetails("Tasks")]}
            {#ix-set:AttributeName = "<#Read axis info task#>"}
            AxoReadAxisInfo_Task                    :   AXOpen.Core.AxoToggleTask;
            {#ix-attr:[ComponentDetails("Tasks")]}
            {#ix-set:AttributeName = "<#Read axis info valid#>"}
            AxoReadAxisInfo_Valid                   :   BOOL;
            {#ix-attr:[ComponentDetails("Tasks")]}
            {#ix-set:AttributeName = "<#Read axis info busy#>"}
            AxoReadAxisInfo_Busy                    :   BOOL;
            {#ix-attr:[ComponentDetails("Tasks")]}
            {#ix-set:AttributeName = "<#Read axis info error#>"}
            AxoReadAxisInfo_Error                   :   BOOL;
            {#ix-attr:[ComponentDetails("Tasks")]}
            {#ix-set:AttributeName = "<#Read axis info error ID#>"}
            AxoReadAxisInfo_ErrorID                 :   WORD;
            {#ix-attr:[ComponentDetails("Tasks")]}
            {#ix-set:AttributeName = "<#Read axis info home absolute switch#>"}
            AxoReadAxisInfo_HomeAbsSwitch           :   BOOL;
            {#ix-attr:[ComponentDetails("Tasks")]}
            {#ix-set:AttributeName = "<#Read axis info limit switch positive#>"}
            AxoReadAxisInfo_LimitSwitchPos          :   BOOL;
            {#ix-attr:[ComponentDetails("Tasks")]}
            {#ix-set:AttributeName = "<#Read axis info limit switch negative#>"}
            AxoReadAxisInfo_LimitSwitchNeg          :   BOOL;
            {#ix-attr:[ComponentDetails("Tasks")]}
            {#ix-set:AttributeName = "<#Read axis info simulation#>"}
            AxoReadAxisInfo_Simulation              :   BOOL;
            {#ix-attr:[ComponentDetails("Tasks")]}
            {#ix-set:AttributeName = "<#Read axis info communication ready#>"}
            AxoReadAxisInfo_CommunicationReady      :   BOOL;
            {#ix-attr:[ComponentDetails("Tasks")]}
            {#ix-set:AttributeName = "<#Read axis info ready for power on#>"}
            AxoReadAxisInfo_ReadyForPowerOn         :   BOOL;
            {#ix-attr:[ComponentDetails("Tasks")]}
            {#ix-set:AttributeName = "<#Read axis info power on#>"}
            AxoReadAxisInfo_PowerOn                 :   BOOL;
            {#ix-attr:[ComponentDetails("Tasks")]}
            {#ix-set:AttributeName = "<#Read axis info is homed#>"}
            AxoReadAxisInfo_IsHomed                 :   BOOL;
            {#ix-attr:[ComponentDetails("Tasks")]}
            {#ix-set:AttributeName = "<#Read axis info warning#>"}
            AxoReadAxisInfo_AxisWarning             :   BOOL;
            //***********ReadAxisError************************
            {#ix-attr:[Container(Layout.UniformGrid)]}
            {#ix-attr:[Group(GroupLayout.GroupBox)]}
            {#ix-attr:[ComponentDetails("Tasks")]}
            {#ix-set:AttributeName = "<#Read axis error task#>"}
            AxoReadAxisError_Task                   :   AXOpen.Core.AxoToggleTask;
            {#ix-attr:[ComponentDetails("Tasks")]}
            {#ix-set:AttributeName = "<#Read axis error valid#>"}
            AxoReadAxisError_Valid                  :   BOOL;
            {#ix-attr:[ComponentDetails("Tasks")]}
            {#ix-set:AttributeName = "<#Read axis error busy#>"}
            AxoReadAxisError_Busy                   :   BOOL;
            {#ix-attr:[ComponentDetails("Tasks")]}
            {#ix-set:AttributeName = "<#Read axis error error#>"}
            AxoReadAxisError_Error                  :   BOOL;
            {#ix-attr:[ComponentDetails("Tasks")]}
            {#ix-set:AttributeName = "<#Read axis error error ID#>"}
            AxoReadAxisError_ErrorID                :   WORD;
            {#ix-attr:[ComponentDetails("Tasks")]}
            {#ix-set:AttributeName = "<#Read axis error axis error ID#>"}
            AxoReadAxisError_AxisErrorID            :   WORD;
            //***********Reset********************************
            {#ix-attr:[Container(Layout.UniformGrid)]}
            {#ix-attr:[Group(GroupLayout.GroupBox)]}
            {#ix-attr:[ComponentDetails("Tasks")]}
            {#ix-set:AttributeName = "<#Reset task#>"}
            AxoReset_Task                           :   AXOpen.Core.AxoTask;
            {#ix-attr:[ComponentDetails("Tasks")]}
            {#ix-set:AttributeName = "<#Reset done#>"}
            AxoReset_Done                           :   BOOL;
            {#ix-attr:[ComponentDetails("Tasks")]}
            {#ix-set:AttributeName = "<#Reset busy#>"}
            AxoReset_Busy                           :   BOOL;
            {#ix-attr:[ComponentDetails("Tasks")]}
            {#ix-set:AttributeName = "<#Reset error#>"}
            AxoReset_Error                          :   BOOL;
            {#ix-attr:[ComponentDetails("Tasks")]}
            {#ix-set:AttributeName = "<#Reset error ID#>"}
            AxoReset_ErrorID                        :   WORD;
            //***********Jog**********************************
            {#ix-attr:[Container(Layout.UniformGrid)]}
            {#ix-attr:[Group(GroupLayout.GroupBox)]}
            {#ix-attr:[ComponentDetails("Tasks")]}
            {#ix-set:AttributeName = "<#Jog positive#>"}
            AxoJogPositive                          :   AXOpen.Components.Abstractions.AxoDrives.AxoMotionJogTask;
            {#ix-attr:[ComponentDetails("Tasks")]}
            {#ix-set:AttributeName = "<#Jog negative#>"}
            AxoJogNegative                          :   AXOpen.Components.Abstractions.AxoDrives.AxoMotionJogTask;
            {#ix-attr:[ComponentDetails("Tasks")]}
            {#ix-set:AttributeName = "<#Jog velocity#>"}
            AxoJog_Velocity                         :   LREAL;
            {#ix-attr:[ComponentDetails("Tasks")]}
            {#ix-set:AttributeName = "<#Jog acceleration#>"}
            AxoJog_Acceleration                     :   LREAL;
            {#ix-attr:[ComponentDetails("Tasks")]}
            {#ix-set:AttributeName = "<#Jog deceleration#>"}
            AxoJog_Deceleration                     :   LREAL;
            {#ix-attr:[ComponentDetails("Tasks")]}
            {#ix-set:AttributeName = "<#Jog jerk#>"}
            AxoJog_Jerk                             :   LREAL;
            {#ix-attr:[ComponentDetails("Tasks")]}
            {#ix-set:AttributeName = "<#Jog direction#>"}
            AxoJog_Direction                        :   AXOpen.Components.Abstractions.AxoDrives.eAxoDriveDirection;
            {#ix-attr:[ComponentDetails("Tasks")]}
            {#ix-set:AttributeName = "<#Jog velocity#>"}
            AxoJogInVelocity                        :   BOOL;
            {#ix-attr:[ComponentDetails("Tasks")]}
            {#ix-set:AttributeName = "<#Jog active#>"}
            AxoJog_Active                           :   BOOL;
            {#ix-attr:[ComponentDetails("Tasks")]}
            {#ix-set:AttributeName = "<#Jog done#>"}
            AxoJog_Done                             :   BOOL;
            {#ix-attr:[ComponentDetails("Tasks")]}
            {#ix-set:AttributeName = "<#Jog busy#>"}
            AxoJog_Busy                             :   BOOL;
            {#ix-attr:[ComponentDetails("Tasks")]}
            {#ix-set:AttributeName = "<#Jog error#>"}
            AxoJog_Error                            :   BOOL;
            {#ix-attr:[ComponentDetails("Tasks")]}
            {#ix-set:AttributeName = "<#Jog error ID#>"}
            AxoJog_ErrorID                          :   WORD;
            {#ix-attr:[ComponentDetails("Tasks")]}
            {#ix-set:AttributeName = "<#Jog aborted#>"}
            AxoJog_CommandAborted                   :   BOOL;
        END_VAR

        VAR PRIVATE
            _AxisRef                                :   AXOpen.Components.Abstractions.AxoDrives.AxoAxisRef;
            _movementDisabled                       :   BOOL;
            //***********Stop*********************************
            _AxoStop_Deceleration                   :   LREAL;
            _AxoStop_Jerk                           :   LREAL;
            //***********Halt*********************************
            _AxoHalt_Deceleration                   :   LREAL;
            _AxoHalt_Jerk                           :   LREAL;
            //***********Home*********************************
            _AxoHome_Position                       :   LREAL;
            _AxoHome_HommingMode                    :   INT;
            _AxoHome_Velocity                       :   LREAL;
            _AxoHome_Acceleration                   :   LREAL;
            _AxoHome_Deceleration                   :   LREAL;
            //***********MoveAbsolute*************************
            _AxoMoveAbsolute_ContinuousUpdate       :   BOOL;
            _AxoMoveAbsolute_Position               :   LREAL;
            _AxoMoveAbsolute_Velocity               :   LREAL;
            _AxoMoveAbsolute_Acceleration           :   LREAL;
            _AxoMoveAbsolute_Deceleration           :   LREAL;
            _AxoMoveAbsolute_Jerk                   :   LREAL;
            _AxoMoveAbsolute_Direction              :   AXOpen.Components.Abstractions.AxoDrives.eAxoDriveDirection;
            //***********MoveRelative*************************
            _AxoMoveRelative_ContinuousUpdate       :   BOOL;
            _AxoMoveRelative_Distance               :   LREAL;
            _AxoMoveRelative_Velocity               :   LREAL;
            _AxoMoveRelative_Acceleration           :   LREAL;
            _AxoMoveRelative_Deceleration           :   LREAL;
            _AxoMoveRelative_Jerk                   :   LREAL;
            _AxoMoveRelative_Direction              :   AXOpen.Components.Abstractions.AxoDrives.eAxoDriveDirection;
            //***********MoveAdditive*************************
            _AxoMoveAdditive_ContinuousUpdate       :   BOOL;
            _AxoMoveAdditive_Distance               :   LREAL;
            _AxoMoveAdditive_Velocity               :   LREAL;
            _AxoMoveAdditive_Acceleration           :   LREAL;
            _AxoMoveAdditive_Deceleration           :   LREAL;
            _AxoMoveAdditive_Jerk                   :   LREAL;
            _AxoMoveAdditive_Direction              :   AXOpen.Components.Abstractions.AxoDrives.eAxoDriveDirection;
            //***********MoveVelocity*************************
            _AxoMoveVelocity_ContinuousUpdate       :   BOOL;
            _AxoMoveVelocity_Velocity               :   LREAL;
            _AxoMoveVelocity_Acceleration           :   LREAL;
            _AxoMoveVelocity_Deceleration           :   LREAL;
            _AxoMoveVelocity_Jerk                   :   LREAL;
            _AxoMoveVelocity_Direction              :   AXOpen.Components.Abstractions.AxoDrives.eAxoDriveDirection;
            //***********TorqueControl************************
            _AxoTorqueControl_ContinuousUpdate      :   BOOL;
            _AxoTorqueControl_Torque                :   LREAL;
            _AxoTorqueControl_TorqueRamp            :   LREAL;
            _AxoTorqueControl_Velocity              :   LREAL;
            _AxoTorqueControl_Acceleration          :   LREAL;
            _AxoTorqueControl_Deceleration          :   LREAL;
            _AxoTorqueControl_Jerk                  :   LREAL;
            _AxoTorqueControl_Direction             :   AXOpen.Components.Abstractions.AxoDrives.eAxoDriveDirection;
            //***********SetPosition**************************
            _AxoSetPosition_Position                :   REAL;
            _AxoSetPosition_Relative                :   BOOL;
            _AxoSetPosition_ExecutionMode           :   AXOpen.Components.Abstractions.AxoDrives.eAxoExecutionMode;
            //***********SetOverride**************************
            _AxoSetOverride_VelFactor               :   LREAL;
            _AxoSetOverride_AccFactor               :   LREAL;
            _AxoSetOverride_JerkFactor              :   LREAL;
            //***********ReadParameter************************
            _AxoReadParameter_ParameterNumber       :   INT;
            //***********ReadBoolParameter********************
            _AxoReadBoolParameter_ParameterNumber   :   INT;
            //***********WriteParameter***********************
            _AxoWriteParameter_ParameterNumber      :   INT;
            _AxoWriteParameter_Value                :   REAL;
            _AxoWriteParameter_ExecutionMode        :   AXOpen.Components.Abstractions.AxoDrives.eAxoExecutionMode;
            //***********WriteBoolParameter*******************
            _AxoWriteBoolParameter_ParameterNumber  :   INT;
            _AxoWriteBoolParameter_Value            :   BOOL;
            _AxoWriteBoolParameter_ExecutionMode    :   AXOpen.Components.Abstractions.AxoDrives.eAxoExecutionMode;
            //***********ReadDigitalInput*********************
            _AxoReadDigitalInput_InputNumber        :   INT;
            //***********ReadDigitalOutput********************
            _AxoReadDigitalOutput_OutputNumber      :   INT;
            //***********WriteDigitalOutput*******************
            _AxoWriteDigitalOutput_OutputNumber     :   INT;
            _AxoWriteDigitalOutput_Value            :   BOOL;
            _AxoWriteDigitalOutput_ExecutionMode    :   AXOpen.Components.Abstractions.AxoDrives.eAxoExecutionMode;
            //***********ReadMotionState**********************
            _AxoReadMotionState_Source              :   AXOpen.Components.Abstractions.AxoDrives.eAxoSource;
            //***********Jog**********************************
            _AxoJog_Velocity                        :   LREAL;
            _AxoJog_Acceleration                    :   LREAL;
            _AxoJog_Deceleration                    :   LREAL;
            _AxoJog_Jerk                            :   LREAL;
            _AxoJog_Direction                       :   AXOpen.Components.Abstractions.AxoDrives.eAxoDriveDirection;
            _AxoJogInVelocity                       :   BOOL;
            _AxoJog_Active                          :   BOOL;
        END_VAR

        ///<summary>
        /// Runs tasks and logic of this component.
        /// >[!IMPORTANT] This method or one of its overloads must be called cyclically.
        ///</summary>
        METHOD PUBLIC Run
            VAR_INPUT
                parent          :   IAxoObject;
                refAxisIn       :   REF_TO  ARRAY[*] OF BYTE;   //  Reference to the input data of the axis
                refAxisOut      :   REF_TO  ARRAY[*] OF BYTE;   //  Reference to the output data of the axis
                Enable          :   BOOL;                       //  As long as ‘Enable’ is true, power is being enabled.
                EnablePositive  :   BOOL;                       //  As long as ‘Enable’ is true, this permits motion in positive direction
                EnableNegative  :   BOOL;                       //  As long as ‘Enable’ is true, this permits motion in negative direction
            END_VAR
            IF parent = NULL THEN
                DriveStatus.Error.Id := UINT#700; //_CurrentMotionTaskId
                RETURN;
            END_IF;

            Messenger.ActivateOnCondition(ULINT#700,parent = NULL, eAxoMessageCategory#ProgrammingError);

            IF NOT THIS.IsValidReferences(refAxisIn,refAxisOut) THEN
                RETURN;
            END_IF;

            THIS.Initialize(parent);
            THIS.Open();
            THIS.UpdateInputs(refAxisIn,_AxisRef);
            THIS.Execute(_AxisRef,Enable,EnablePositive,EnableNegative);
            THIS.UpdateOutputs(_AxisRef,refAxisIn);
            THIS.Close();
        END_METHOD

        ///<summary>
        /// Runs tasks and logic of this component.
        /// >[!IMPORTANT] This method or one of its overloads must be called cyclically.
        ///</summary>
        METHOD PUBLIC Run
            VAR_INPUT
                parent          :   IAxoContext;
                refAxisIn       :   REF_TO  ARRAY[*] OF BYTE;   //  Reference to the input data of the axis
                refAxisOut      :   REF_TO  ARRAY[*] OF BYTE;   //  Reference to the output data of the axis
                Enable          :   BOOL;                       //  As long as ‘Enable’ is true, power is being enabled.
                EnablePositive  :   BOOL;                       //  As long as ‘Enable’ is true, this permits motion in positive direction
                EnableNegative  :   BOOL;                       //  As long as ‘Enable’ is true, this permits motion in negative direction
            END_VAR
            IF parent = NULL THEN
                DriveStatus.Error.Id := UINT#700;
                RETURN;
            END_IF;

            Messenger.ActivateOnCondition(ULINT#700,parent = NULL, eAxoMessageCategory#ProgrammingError);

            IF NOT THIS.IsValidReferences(refAxisIn,refAxisOut) THEN
                RETURN;
            END_IF;

            THIS.Initialize(parent);
            THIS.Open();
            THIS.UpdateInputs(refAxisIn,_AxisRef);
            THIS.Execute(_AxisRef,Enable,EnablePositive,EnableNegative);
            THIS.UpdateOutputs(_AxisRef,refAxisIn);
            THIS.Close();
        END_METHOD

        METHOD PRIVATE Execute
            VAR_IN_OUT
                AxisRef :   AxoAxisRef;
            END_VAR
            VAR_INPUT
                Enable          :   BOOL;                       //  As long as ‘Enable’ is true, power is being enabled.
                EnablePositive  :   BOOL;                       //  As long as ‘Enable’ is true, this permits motion in positive direction
                EnableNegative  :   BOOL;                       //  As long as ‘Enable’ is true, this permits motion in negative direction
            END_VAR

            Messenger.Serve(THIS);

            AxoPower_Task.Initialize(THIS);
            AxoStop_Task.Initialize(THIS);
            AxoHalt_Task.Initialize(THIS);
            AxoHome_Task.Initialize(THIS);
            AxoMoveAbsolute_Task.Initialize(THIS);
            AxoMoveRelative_Task.Initialize(THIS);
            AxoMoveAdditive_Task.Initialize(THIS);
            AxoMoveVelocity_Task.Initialize(THIS);
            AxoTorqueControl_Task.Initialize(THIS);
            AxoSetPosition_Task.Initialize(THIS);
            AxoSetOverride_Task.Initialize(THIS);
            AxoReadParameter_Task.Initialize(THIS);
            AxoReadBoolParameter_Task.Initialize(THIS);
            AxoWriteParameter_Task.Initialize(THIS);
            AxoWriteBoolParameter_Task.Initialize(THIS);
            AxoReadDigitalInput_Task.Initialize(THIS);
            AxoReadDigitalOutput_Task.Initialize(THIS);
            AxoWriteDigitalOutput_Task.Initialize(THIS);
            AxoReadActualPosition_Task.Initialize(THIS);
            AxoReadActualVelocity_Task.Initialize(THIS);
            AxoReadActualTorque_Task.Initialize(THIS);
            AxoReadStatus_Task.Initialize(THIS);
            AxoReadMotionState_Task.Initialize(THIS);
            AxoReadAxisInfo_Task.Initialize(THIS);
            AxoReadAxisError_Task.Initialize(THIS);
            AxoReset_Task.Initialize(THIS);
            AxoJogPositive.Initialize(THIS);
            AxoJogNegative.Initialize(THIS);

            //*************AXO_POWER********************
            AxoPower_Task.Run(Enable,EnablePositive,EnableNegative);
            THIS.MC_Power(AxisRef,
                          AxoPower_Task.IsSwitchedOn(),
                          AxoPower_Status,
                          AxoPower_Valid,
                          AxoPower_Error,
                          AxoPower_ErrorID);
            Messenger.ActivateOnCondition(TO_ULINT(AxoPower_ErrorID),AxoPower_Error,eAxoMessageCategory#Error);
            //******************************************
            _movementDisabled := NOT AxoPower_Status;
            //*************AXO_STOP*********************
            AxoStop_Task.SetIsDisabled(FALSE);
            THIS.MC_Stop(AxisRef,
                        AxoStop_Task.Execute() OR AxoStop_Task.IsDone() AND AxoStop_Task.IsInvokeCalled(),
                        _AxoStop_Deceleration,
                        _AxoStop_Jerk,
                        AxoStop_Done,
                        AxoStop_Busy,
                        AxoStop_Active,
                        AxoStop_CommandAborted,
                        AxoStop_Error,
                        AxoStop_ErrorID);
            Messenger.ActivateOnCondition(TO_ULINT(AxoStop_ErrorID),AxoStop_Error,eAxoMessageCategory#Error);
            //******************************************
            _movementDisabled := _movementDisabled OR AxoStop_Active OR AxoStop_Task.IsDone() AND AxoStop_Task.IsInvokeCalled();
            //*************AXO_HALT*********************
            AxoHalt_Task.SetIsDisabled(FALSE);
            THIS.MC_Halt(AxisRef,
                        AxoHalt_Task.Execute(),
                        _AxoHalt_Deceleration,
                        _AxoHalt_Jerk,
                        AxoHalt_Done,
                        AxoHalt_Busy,
                        AxoHalt_Active,
                        AxoHalt_CommandAborted,
                        AxoHalt_Error,
                        AxoHalt_ErrorID);

                        IF AxoHalt_Task.Execute() THEN
                            AxoHalt_Task.DoneWhen(AxoHalt_Done);
                            AxoHalt_Task.ThrowWhen(AxoHalt_Error,CONCAT('MC_Halt has thrown an error: ', ToString(AxoHalt_ErrorID)));
                            IF AxoHalt_CommandAborted THEN
                                AxoHalt_Task.Abort();
                            END_IF;
                        END_IF;
            Messenger.ActivateOnCondition(TO_ULINT(AxoHalt_ErrorID),AxoHalt_Error,eAxoMessageCategory#Error);
            //******************************************
            _movementDisabled := _movementDisabled OR AxoHalt_Active;

            //*************AXO_HOME*********************
            AxoHome_Task.SetIsDisabled(_movementDisabled);
            THIS.MC_Home(AxisRef,
                        AxoHome_Task.Execute(),
                        _AxoHome_Position,
                        _AxoHome_HommingMode,
                        _AxoHome_Velocity,
                        _AxoHome_Acceleration,
                        _AxoHome_Deceleration,
                        AxoHome_Done,
                        AxoHome_Busy,
                        AxoHome_Active,
                        AxoHome_CommandAborted,
                        AxoHome_Error,
                        AxoHome_ErrorID);

            IF AxoHome_Task.Execute() THEN
                AxoHome_Task.DoneWhen(AxoHome_Done);
                AxoHome_Task.ThrowWhen(AxoHome_Error,CONCAT('MC_Home has thrown an error: ', ToString(AxoHome_ErrorID)));
                IF AxoHome_CommandAborted THEN
                    AxoHome_Task.Abort();
                END_IF;
            END_IF;
            Messenger.ActivateOnCondition(TO_ULINT(AxoHome_ErrorID),AxoHome_Error,eAxoMessageCategory#Error);
            //******************************************

            //*************AXO_MOVE_ABSOLUTE************
            AxoMoveAbsolute_Task.SetIsDisabled(_movementDisabled); //TODO Enable negative positive
            THIS.MC_MoveAbsolute(AxisRef,
                        AxoMoveAbsolute_Task.Execute(),
                        _AxoMoveAbsolute_ContinuousUpdate,
                        _AxoMoveAbsolute_Position,
                        _AxoMoveAbsolute_Velocity,
                        _AxoMoveAbsolute_Acceleration,
                        _AxoMoveAbsolute_Deceleration,
                        _AxoMoveAbsolute_Jerk,
                        _AxoMoveAbsolute_Direction,
                        AxoMoveAbsolute_Done,
                        AxoMoveAbsolute_Busy,
                        AxoMoveAbsolute_Active,
                        AxoMoveAbsolute_CommandAborted,
                        AxoMoveAbsolute_Error,
                        AxoMoveAbsolute_ErrorID);

            IF AxoMoveAbsolute_Task.Execute() THEN
                AxoMoveAbsolute_Task.DoneWhen(AxoMoveAbsolute_Done);
                AxoMoveAbsolute_Task.ThrowWhen(AxoMoveAbsolute_Error,CONCAT('MC_MoveAbsolute has thrown an error: ', ToString(AxoMoveAbsolute_ErrorID)));
                IF AxoMoveAbsolute_CommandAborted THEN
                    AxoMoveAbsolute_Task.Abort();
                END_IF;
            END_IF;
            Messenger.ActivateOnCondition(TO_ULINT(AxoMoveAbsolute_ErrorID),AxoMoveAbsolute_Error,eAxoMessageCategory#Error);
            //******************************************

            //*************AXO_MOVE_RELATIVE************
            AxoMoveRelative_Task.SetIsDisabled(_movementDisabled); //TODO Enable negative positive
            THIS.MC_MoveRelative(AxisRef,
                        AxoMoveRelative_Task.Execute(),
                        _AxoMoveRelative_ContinuousUpdate,
                        _AxoMoveRelative_Distance,
                        _AxoMoveRelative_Velocity,
                        _AxoMoveRelative_Acceleration,
                        _AxoMoveRelative_Deceleration,
                        _AxoMoveRelative_Jerk,
                        _AxoMoveRelative_Direction,
                        AxoMoveRelative_Done,
                        AxoMoveRelative_Busy,
                        AxoMoveRelative_Active,
                        AxoMoveRelative_CommandAborted,
                        AxoMoveRelative_Error,
                        AxoMoveRelative_ErrorID);

            IF AxoMoveRelative_Task.Execute() THEN
                AxoMoveRelative_Task.DoneWhen(AxoMoveRelative_Done);
                AxoMoveRelative_Task.ThrowWhen(AxoMoveRelative_Error,CONCAT('MC_MoveRelative has thrown an error: ', ToString(AxoMoveRelative_ErrorID)));
                IF AxoMoveRelative_CommandAborted THEN
                    AxoMoveRelative_Task.Abort();
                END_IF;
            END_IF;
            Messenger.ActivateOnCondition(TO_ULINT(AxoMoveRelative_ErrorID),AxoMoveRelative_Error,eAxoMessageCategory#Error);
            //******************************************

            //*************AXO_MOVE_ADDITIVE************
            AxoMoveAdditive_Task.SetIsDisabled(_movementDisabled); //TODO Enable negative positive
            THIS.MC_MoveAdditive(AxisRef,
                        AxoMoveAdditive_Task.Execute(),
                        _AxoMoveAdditive_ContinuousUpdate,
                        _AxoMoveAdditive_Distance,
                        _AxoMoveAdditive_Velocity,
                        _AxoMoveAdditive_Acceleration,
                        _AxoMoveAdditive_Deceleration,
                        _AxoMoveAdditive_Jerk,
                        _AxoMoveAdditive_Direction,
                        AxoMoveAdditive_Done,
                        AxoMoveAdditive_Busy,
                        AxoMoveAdditive_Active,
                        AxoMoveAdditive_CommandAborted,
                        AxoMoveAdditive_Error,
                        AxoMoveAdditive_ErrorID);

            IF AxoMoveAdditive_Task.Execute() THEN
                AxoMoveAdditive_Task.DoneWhen(AxoMoveAdditive_Done);
                AxoMoveAdditive_Task.ThrowWhen(AxoMoveAdditive_Error,CONCAT('MC_MoveAdditive has thrown an error: ', ToString(AxoMoveAdditive_ErrorID)));
                IF AxoMoveAdditive_CommandAborted THEN
                    AxoMoveAdditive_Task.Abort();
                END_IF;
            END_IF;
            Messenger.ActivateOnCondition(TO_ULINT(AxoMoveAdditive_ErrorID),AxoMoveAdditive_Error,eAxoMessageCategory#Error);
            //******************************************

            //*************AXO_MOVE_VELOCITY************
            AxoMoveVelocity_Task.SetIsDisabled(_movementDisabled); //TODO Enable negative positive
            THIS.MC_MoveVelocity(AxisRef,
                        AxoMoveVelocity_Task.Execute(),
                        _AxoMoveVelocity_ContinuousUpdate,
                        _AxoMoveVelocity_Velocity,
                        _AxoMoveVelocity_Acceleration,
                        _AxoMoveVelocity_Deceleration,
                        _AxoMoveVelocity_Jerk,
                        _AxoMoveVelocity_Direction,
                        AxoMoveVelocity_InVelocity,
                        AxoMoveVelocity_Busy,
                        AxoMoveVelocity_Active,
                        AxoMoveVelocity_CommandAborted,
                        AxoMoveVelocity_Error,
                        AxoMoveVelocity_ErrorID);

            IF AxoMoveVelocity_Task.Execute() THEN
                AxoMoveVelocity_Task.DoneWhen(AxoMoveVelocity_InVelocity);
                AxoMoveVelocity_Task.ThrowWhen(AxoMoveVelocity_Error,CONCAT('MC_MoveVelocity has thrown an error: ', ToString(AxoMoveVelocity_ErrorID)));
                IF AxoMoveVelocity_CommandAborted THEN
                    AxoMoveVelocity_Task.Abort();
                END_IF;
            END_IF;
            Messenger.ActivateOnCondition(TO_ULINT(AxoMoveVelocity_ErrorID),AxoMoveVelocity_Error,eAxoMessageCategory#Error);
            //******************************************

            //*************AXO_TORQUE_CONTROL***********
            AxoTorqueControl_Task.SetIsDisabled(_movementDisabled); //TODO Enable negative positive
            THIS.MC_TorqueControl(AxisRef,
                        AxoTorqueControl_Task.Execute(),
                        _AxoTorqueControl_ContinuousUpdate,
                        _AxoTorqueControl_Torque,
                        _AxoTorqueControl_TorqueRamp,
                        _AxoTorqueControl_Velocity,
                        _AxoTorqueControl_Acceleration,
                        _AxoTorqueControl_Deceleration,
                        _AxoTorqueControl_Jerk,
                        _AxoTorqueControl_Direction,
                        AxoTorqueControl_InTorque,
                        AxoTorqueControl_Busy,
                        AxoTorqueControl_Active,
                        AxoTorqueControl_CommandAborted,
                        AxoTorqueControl_Error,
                        AxoTorqueControl_ErrorID);

            IF AxoTorqueControl_Task.Execute() THEN
                AxoTorqueControl_Task.DoneWhen(AxoTorqueControl_InTorque);
                AxoTorqueControl_Task.ThrowWhen(AxoTorqueControl_Error,CONCAT('MC_TorqueControl has thrown an error: ', ToString(AxoTorqueControl_ErrorID)));
                IF AxoTorqueControl_CommandAborted THEN
                    AxoTorqueControl_Task.Abort();
                END_IF;
            END_IF;
            Messenger.ActivateOnCondition(TO_ULINT(AxoTorqueControl_ErrorID),AxoTorqueControl_Error,eAxoMessageCategory#Error);
            //******************************************

            //*************AXO_SET_POSITION*************
            AxoSetPosition_Task.SetIsDisabled(FALSE);
            THIS.MC_SetPosition(AxisRef,
                        AxoSetPosition_Task.Execute(),
                        _AxoSetPosition_Position,
                        _AxoSetPosition_Relative,
                        _AxoSetPosition_ExecutionMode,
                        AxoSetPosition_Done,
                        AxoSetPosition_Error,
                        AxoSetPosition_ErrorID);

            IF AxoSetPosition_Task.Execute() THEN
                AxoSetPosition_Task.DoneWhen(AxoSetPosition_Done);
                AxoSetPosition_Task.ThrowWhen(AxoSetPosition_Error,CONCAT('MC_SetPosition has thrown an error: ', ToString(AxoSetPosition_ErrorID)));
            END_IF;
            Messenger.ActivateOnCondition(TO_ULINT(AxoSetPosition_ErrorID),AxoSetPosition_Error,eAxoMessageCategory#Error);
            //******************************************

            //*************AXO_SET_OVERRIDE*************
            AxoSetOverride_Task.SetIsDisabled(FALSE);
            THIS.MC_SetOverride(AxisRef,
                        AxoSetOverride_Task.IsSwitchedOn(),
                        _AxoSetOverride_VelFactor,
                        _AxoSetOverride_AccFactor,
                        _AxoSetOverride_JerkFactor,
                        AxoSetOverride_Enabled,
                        AxoSetOverride_Busy,
                        AxoSetOverride_Error,
                        AxoSetOverride_ErrorID);
            Messenger.ActivateOnCondition(TO_ULINT(AxoSetOverride_ErrorID),AxoSetOverride_Error,eAxoMessageCategory#Error);
            //******************************************

            //*************AXO_READ_PARAMETER***********
            AxoReadParameter_Task.SetIsDisabled(FALSE);
            THIS.MC_ReadParameter(AxisRef,
                        AxoReadParameter_Task.IsSwitchedOn(),
                        _AxoReadParameter_ParameterNumber,
                        AxoReadParameter_Valid,
                        AxoReadParameter_Busy,
                        AxoReadParameter_Error,
                        AxoReadParameter_ErrorID,
                        AxoReadParameter_Value);
            Messenger.ActivateOnCondition(TO_ULINT(AxoReadParameter_ErrorID),AxoReadParameter_Error,eAxoMessageCategory#Error);
            //******************************************

            //*************AXO_READ_BOOL_PARAMETER******
            AxoReadBoolParameter_Task.SetIsDisabled(FALSE);
            THIS.MC_ReadBoolParameter(AxisRef,
                        AxoReadBoolParameter_Task.IsSwitchedOn(),
                        _AxoReadBoolParameter_ParameterNumber,
                        AxoReadBoolParameter_Valid,
                        AxoReadBoolParameter_Busy,
                        AxoReadBoolParameter_Error,
                        AxoReadBoolParameter_ErrorID,
                        AxoReadBoolParameter_Value);
            Messenger.ActivateOnCondition(TO_ULINT(AxoReadBoolParameter_ErrorID),AxoReadBoolParameter_Error,eAxoMessageCategory#Error);
            //******************************************

            //*************AXO_WRITE_PARAMETER**********
            AxoWriteParameter_Task.SetIsDisabled(FALSE);
            THIS.MC_WriteParameter(AxisRef,
                        AxoWriteParameter_Task.Execute(),
                        _AxoWriteParameter_ParameterNumber,
                        _AxoWriteParameter_Value,
                        _AxoWriteParameter_ExecutionMode,
                        AxoWriteParameter_Done,
                        AxoWriteParameter_Busy,
                        AxoWriteParameter_Error,
                        AxoWriteParameter_ErrorID);
            Messenger.ActivateOnCondition(TO_ULINT(AxoWriteParameter_ErrorID),AxoWriteParameter_Error,eAxoMessageCategory#Error);
            //******************************************

            //*************AXO_WRITE_BOOL_PARAMETER*****
            AxoWriteBoolParameter_Task.SetIsDisabled(FALSE);
            THIS.MC_WriteBoolParameter(AxisRef,
                        AxoWriteBoolParameter_Task.Execute(),
                        _AxoWriteBoolParameter_ParameterNumber,
                        _AxoWriteBoolParameter_Value,
                        _AxoWriteBoolParameter_ExecutionMode,
                        AxoWriteBoolParameter_Done,
                        AxoWriteBoolParameter_Busy,
                        AxoWriteBoolParameter_Error,
                        AxoWriteBoolParameter_ErrorID);
            Messenger.ActivateOnCondition(TO_ULINT(AxoWriteBoolParameter_ErrorID),AxoWriteBoolParameter_Error,eAxoMessageCategory#Error);
            //******************************************

            //*************AXO_READ_DIGITAL_INPUT*******
            AxoReadDigitalInput_Task.SetIsDisabled(FALSE);
            THIS.MC_ReadDigitalInput(AxisRef,
                        AxoReadDigitalInput_Task.IsSwitchedOn(),
                        _AxoReadDigitalInput_InputNumber,
                        AxoReadDigitalInput_Valid,
                        AxoReadDigitalInput_Busy,
                        AxoReadDigitalInput_Error,
                        AxoReadDigitalInput_ErrorID,
                        AxoReadDigitalInput_Value);
            Messenger.ActivateOnCondition(TO_ULINT(AxoReadDigitalInput_ErrorID),AxoReadDigitalInput_Error,eAxoMessageCategory#Error);
            //******************************************

            //*************AXO_READ_DIGITAL_OUTPUT******
            AxoReadDigitalOutput_Task.SetIsDisabled(FALSE);
            THIS.MC_ReadDigitalInput(AxisRef,
                        AxoReadDigitalOutput_Task.IsSwitchedOn(),
                        _AxoReadDigitalOutput_OutputNumber,
                        AxoReadDigitalOutput_Valid,
                        AxoReadDigitalOutput_Busy,
                        AxoReadDigitalOutput_Error,
                        AxoReadDigitalOutput_ErrorID,
                        AxoReadDigitalOutput_Value);
            Messenger.ActivateOnCondition(TO_ULINT(AxoReadDigitalInput_ErrorID),AxoReadDigitalInput_Error,eAxoMessageCategory#Error);
            //******************************************

            //*************AXO_WRITE_DIGITAL_OUTPUT*****
            AxoWriteDigitalOutput_Task.SetIsDisabled(FALSE);
            THIS.MC_WriteDigitalOutput(AxisRef,
                        AxoWriteDigitalOutput_Task.Execute(),
                        _AxoWriteDigitalOutput_OutputNumber,
                        _AxoWriteDigitalOutput_Value,
                        _AxoWriteDigitalOutput_ExecutionMode,
                        AxoWriteDigitalOutput_Done,
                        AxoWriteDigitalOutput_Busy,
                        AxoWriteDigitalOutput_Error,
                        AxoWriteDigitalOutput_ErrorID);
            Messenger.ActivateOnCondition(TO_ULINT(AxoWriteBoolParameter_ErrorID),AxoWriteBoolParameter_Error,eAxoMessageCategory#Error);
            //******************************************

            //*************AXO_READ_ACTUAL_POSITION*****
            AxoReadActualPosition_Task.SetIsDisabled(FALSE);
            THIS.MC_ReadActualPosition(AxisRef,
                        AxoReadActualPosition_Task.IsSwitchedOn(),
                        AxoReadActualPosition_Valid,
                        AxoReadActualPosition_Busy,
                        AxoReadActualPosition_Error,
                        AxoReadActualPosition_ErrorID,
                        AxoReadActualPosition_Value);
            Messenger.ActivateOnCondition(TO_ULINT(AxoReadActualPosition_ErrorID),AxoReadActualPosition_Error,eAxoMessageCategory#Error);
            //******************************************

            //*************AXO_READ_ACTUAL_VELOCITY*****
            AxoReadActualVelocity_Task.SetIsDisabled(FALSE);
            THIS.MC_ReadActualVelocity(AxisRef,
                        AxoReadActualVelocity_Task.IsSwitchedOn(),
                        AxoReadActualVelocity_Valid,
                        AxoReadActualVelocity_Busy,
                        AxoReadActualVelocity_Error,
                        AxoReadActualVelocity_ErrorID,
                        AxoReadActualVelocity_Value);
            Messenger.ActivateOnCondition(TO_ULINT(AxoReadActualVelocity_ErrorID),AxoReadActualVelocity_Error,eAxoMessageCategory#Error);
            //******************************************

            //*************AXO_READ_ACTUAL_TORQUE*******
            AxoReadActualTorque_Task.SetIsDisabled(FALSE);
            THIS.MC_ReadActualTorque(AxisRef,
                        AxoReadActualTorque_Task.IsSwitchedOn(),
                        AxoReadActualTorque_Valid,
                        AxoReadActualTorque_Busy,
                        AxoReadActualTorque_Error,
                        AxoReadActualTorque_ErrorID,
                        AxoReadActualTorque_Value);
            Messenger.ActivateOnCondition(TO_ULINT(AxoReadActualTorque_ErrorID),AxoReadActualTorque_Error,eAxoMessageCategory#Error);
            //******************************************

            //*************AXO_READ_STATUS**************
            AxoReadStatus_Task.SetIsDisabled(FALSE);
            THIS.MC_ReadStatus(AxisRef,
                        AxoReadStatus_Task.IsSwitchedOn(),
                        AxoReadStatus_Valid,
                        AxoReadStatus_Busy,
                        AxoReadStatus_Error,
                        AxoReadStatus_ErrorID,
                        AxoReadStatus_ErrorStop,
                        AxoReadStatus_Disabled,
                        AxoReadStatus_Stopping,
                        AxoReadStatus_Homing,
                        AxoReadStatus_Standstill,
                        AxoReadStatus_DiscreteMotion,
                        AxoReadStatus_ContinuousMotion,
                        AxoReadStatus_SynchronizedMotion);
            Messenger.ActivateOnCondition(TO_ULINT(AxoReadStatus_ErrorID),AxoReadStatus_Error,eAxoMessageCategory#Error);
            //******************************************

            //*************AXO_READ_MOTION_STATE********
            AxoReadMotionState_Task.SetIsDisabled(FALSE);
            THIS.MC_ReadMotionState(AxisRef,
                        AxoReadMotionState_Task.IsSwitchedOn(),
                        _AxoReadMotionState_Source,
                        AxoReadMotionState_Valid,
                        AxoReadMotionState_Busy,
                        AxoReadMotionState_Error,
                        AxoReadMotionState_ErrorID,
                        AxoReadMotionState_ConstantVelocity,
                        AxoReadMotionState_Accelerating,
                        AxoReadMotionState_Decelerating,
                        AxoReadMotionState_DirectionPositive,
                        AxoReadMotionState_DirectionNegative);
            Messenger.ActivateOnCondition(TO_ULINT(AxoReadMotionState_ErrorID),AxoReadMotionState_Error,eAxoMessageCategory#Error);
            //******************************************

            //*************AXO_READ_AXIS_INFO***********
            AxoReadAxisInfo_Task.SetIsDisabled(FALSE);
            THIS.MC_ReadAxisInfo(AxisRef,
                        AxoReadAxisInfo_Task.IsSwitchedOn(),
                        AxoReadAxisInfo_Valid,
                        AxoReadAxisInfo_Busy,
                        AxoReadAxisInfo_Error,
                        AxoReadAxisInfo_ErrorID,
                        AxoReadAxisInfo_HomeAbsSwitch,
                        AxoReadAxisInfo_LimitSwitchPos,
                        AxoReadAxisInfo_LimitSwitchNeg,
                        AxoReadAxisInfo_Simulation,
                        AxoReadAxisInfo_CommunicationReady,
                        AxoReadAxisInfo_ReadyForPowerOn,
                        AxoReadAxisInfo_PowerOn,
                        AxoReadAxisInfo_IsHomed,
                        AxoReadAxisInfo_AxisWarning);
            Messenger.ActivateOnCondition(TO_ULINT(AxoReadAxisInfo_ErrorID),AxoReadAxisInfo_Error,eAxoMessageCategory#Error);
            //******************************************

            //*************AXO_READ_AXIS_ERROR**********
            AxoReadAxisError_Task.SetIsDisabled(FALSE);
            THIS.MC_ReadAxisError(AxisRef,
                        AxoReadAxisError_Task.IsSwitchedOn(),
                        AxoReadAxisError_Valid,
                        AxoReadAxisError_Busy,
                        AxoReadAxisError_Error,
                        AxoReadAxisError_ErrorID,
                        AxoReadAxisError_AxisErrorID);
                        Messenger.ActivateOnCondition(TO_ULINT(AxoReadAxisError_ErrorID),AxoReadAxisError_Error,eAxoMessageCategory#Error);
            //******************************************

            //*************AXO_RESET********************
            AxoReset_Task.SetIsDisabled(FALSE);
            THIS.MC_Reset(AxisRef,
                        AxoReset_Task.Execute(),
                        AxoReset_Done,
                        AxoReset_Busy,
                        AxoReset_Error,
                        AxoReset_ErrorID);
            Messenger.ActivateOnCondition(TO_ULINT(AxoReset_ErrorID),AxoReset_Error,eAxoMessageCategory#Error);
            //******************************************

            //*************AXO_JOG**********************
            AxoJogPositive.SetIsDisabled(_movementDisabled OR NOT EnablePositive OR AxoJogNegative.IsSwitchedOn());
            AxoJogNegative.SetIsDisabled(_movementDisabled OR NOT EnableNegative OR AxoJogPositive.IsSwitchedOn());
            IF AxoJogPositive.IsSwitchedOn() THEN
                _AxoJog_Direction := AXOpen.Components.Abstractions.AxoDrives.eAxoDriveDirection#PositiveDirection;
            ELSIF AxoJogNegative.IsSwitchedOn() THEN
                _AxoJog_Direction := AXOpen.Components.Abstractions.AxoDrives.eAxoDriveDirection#NegativeDirection;
            END_IF;
            IF AxoJogPositive.IsSwitchedOn() OR AxoJogNegative.IsSwitchedOn() THEN
                IF AxoJogPositive.StartMotion OR AxoJogNegative.StartMotion THEN
                    AxoJogPositive.StartMotion := FALSE;
                    AxoJogNegative.StartMotion := FALSE;
                END_IF;
                THIS.AxoMoveVelocity(FALSE,
                                    _AxoJog_Velocity,
                                    _AxoJog_Acceleration,
                                    _AxoJog_Deceleration,
                                    _AxoJog_Jerk,
                                    _AxoJog_Direction);
            ELSIF AxoJogPositive.StopMotion OR AxoJogNegative.StopMotion THEN
                THIS.AxoMoveVelocity(FALSE);
                THIS.AxoHalt(_AxoJog_Deceleration,_AxoJog_Jerk);
                AxoJogPositive.StopMotion := FALSE;
                AxoJogNegative.StopMotion := FALSE;
            END_IF;
            //******************************************
        END_METHOD

        ///<summary>
		/// Restores this instance .
        ///</summary>
        METHOD PROTECTED OVERRIDE Restore: IAxoTask
            VAR
                _index : INT;
            END_VAR
            // Status.Action.Id := UINT#0;
            // Status.Error.Id  := UINT#0;
            Messenger.Restore();
            TaskMessenger.Restore();

            // AxoPower_Task.Restore();
            AxoStop_Task.Restore();
            AxoHalt_Task.Restore();
            AxoHome_Task.Restore();
            AxoMoveAbsolute_Task.Restore();
            AxoMoveRelative_Task.Restore();
            AxoMoveAdditive_Task.Restore();
            AxoMoveVelocity_Task.Restore();
            AxoTorqueControl_Task.Restore();
            AxoSetPosition_Task.Restore();
            AxoSetOverride_Task.SwitchOff();
            AxoReadParameter_Task.SwitchOff();
            AxoReadBoolParameter_Task.SwitchOff();
            AxoWriteParameter_Task.Restore();
            AxoWriteBoolParameter_Task.Restore();
            AxoReadDigitalInput_Task.SwitchOff();
            AxoReadDigitalOutput_Task.SwitchOff();
            AxoWriteDigitalOutput_Task.Restore();
            AxoReadActualPosition_Task.SwitchOff();
            AxoReadActualVelocity_Task.SwitchOff();
            AxoReadActualTorque_Task.SwitchOff();
            AxoReadStatus_Task.SwitchOff();
            AxoReadMotionState_Task.SwitchOff();
            AxoReadAxisInfo_Task.SwitchOff();
            AxoReadAxisError_Task.SwitchOff();
            AxoReset_Task.Restore();
            // AxoJogPositive.Restore();
            // AxoJogNegative.Restore();

            RestoreTask.DoneWhen(TRUE);
        END_METHOD

        ///<summary>
		/// Custom logic for the manual control.
        ///</summary>
        METHOD PROTECTED OVERRIDE ManualControl
            //***********Stop*********************************
            _AxoStop_Deceleration                   := AxoStop_Deceleration;
            _AxoStop_Jerk                           := AxoStop_Jerk;
            //***********Halt*********************************
            _AxoHalt_Deceleration                   := AxoHalt_Deceleration;
            _AxoHalt_Jerk                           := AxoHalt_Jerk;
            //***********Home*********************************
            _AxoHome_Position                       := AxoHome_Position;
            _AxoHome_HommingMode                    := AxoHome_HommingMode;
            _AxoHome_Velocity                       := AxoHome_Velocity;
            _AxoHome_Acceleration                   := AxoHome_Acceleration;
            _AxoHome_Deceleration                   := AxoHome_Deceleration;
            //***********MoveAbsolute*************************
            _AxoMoveAbsolute_ContinuousUpdate       := AxoMoveAbsolute_ContinuousUpdate;
            _AxoMoveAbsolute_Position               := AxoMoveAbsolute_Position;
            _AxoMoveAbsolute_Velocity               := AxoMoveAbsolute_Velocity;
            _AxoMoveAbsolute_Acceleration           := AxoMoveAbsolute_Acceleration;
            _AxoMoveAbsolute_Deceleration           := AxoMoveAbsolute_Deceleration;
            _AxoMoveAbsolute_Jerk                   := AxoMoveAbsolute_Jerk;
            _AxoMoveAbsolute_Direction              := AxoMoveAbsolute_Direction;
            //***********MoveRelative*************************
            _AxoMoveRelative_ContinuousUpdate       := AxoMoveRelative_ContinuousUpdate;
            _AxoMoveRelative_Distance               := AxoMoveRelative_Distance;
            _AxoMoveRelative_Velocity               := AxoMoveRelative_Velocity;
            _AxoMoveRelative_Acceleration           := AxoMoveRelative_Acceleration;
            _AxoMoveRelative_Deceleration           := AxoMoveRelative_Deceleration;
            _AxoMoveRelative_Jerk                   := AxoMoveRelative_Jerk;
            _AxoMoveRelative_Direction              := AxoMoveRelative_Direction;
            //***********MoveAdditive*************************
            _AxoMoveAdditive_ContinuousUpdate       := AxoMoveAdditive_ContinuousUpdate;
            _AxoMoveAdditive_Distance               := AxoMoveAdditive_Distance;
            _AxoMoveAdditive_Velocity               := AxoMoveAdditive_Velocity;
            _AxoMoveAdditive_Acceleration           := AxoMoveAdditive_Acceleration;
            _AxoMoveAdditive_Deceleration           := AxoMoveAdditive_Deceleration;
            _AxoMoveAdditive_Jerk                   := AxoMoveAdditive_Jerk;
            _AxoMoveAdditive_Direction              := AxoMoveAdditive_Direction;
            //***********MoveVelocity*************************
            _AxoMoveVelocity_ContinuousUpdate       := AxoMoveVelocity_ContinuousUpdate;
            _AxoMoveVelocity_Velocity               := AxoMoveVelocity_Velocity;
            _AxoMoveVelocity_Acceleration           := AxoMoveVelocity_Acceleration;
            _AxoMoveVelocity_Deceleration           := AxoMoveVelocity_Deceleration;
            _AxoMoveVelocity_Jerk                   := AxoMoveVelocity_Jerk;
            _AxoMoveVelocity_Direction              := AxoMoveVelocity_Direction;
            //***********TorqueControl************************
            _AxoTorqueControl_ContinuousUpdate      := AxoTorqueControl_ContinuousUpdate;
            _AxoTorqueControl_Torque                := AxoTorqueControl_Torque;
            _AxoTorqueControl_TorqueRamp            := AxoTorqueControl_TorqueRamp;
            _AxoTorqueControl_Velocity              := AxoTorqueControl_Velocity;
            _AxoTorqueControl_Acceleration          := AxoTorqueControl_Acceleration;
            _AxoTorqueControl_Deceleration          := AxoTorqueControl_Deceleration;
            _AxoTorqueControl_Jerk                  := AxoTorqueControl_Jerk;
            _AxoTorqueControl_Direction             := AxoTorqueControl_Direction;
            //***********SetPosition**************************
            _AxoSetPosition_Position                := AxoSetPosition_Position;
            _AxoSetPosition_Relative                := AxoSetPosition_Relative;
            _AxoSetPosition_ExecutionMode           := AxoSetPosition_ExecutionMode;
            //***********SetOverride**************************
            _AxoSetOverride_VelFactor               := AxoSetOverride_VelFactor;
            _AxoSetOverride_AccFactor               := AxoSetOverride_AccFactor;
            _AxoSetOverride_JerkFactor              := AxoSetOverride_JerkFactor;
            //***********ReadParameter************************
            _AxoReadParameter_ParameterNumber       := AxoReadParameter_ParameterNumber;
            //***********ReadBoolParameter********************
            _AxoReadBoolParameter_ParameterNumber   := AxoReadBoolParameter_ParameterNumber;
            //***********WriteParameter***********************
            _AxoWriteParameter_ParameterNumber      := AxoWriteParameter_ParameterNumber;
            _AxoWriteParameter_Value                := AxoWriteParameter_Value;
            _AxoWriteParameter_ExecutionMode        := AxoWriteParameter_ExecutionMode;
            //***********WriteBoolParameter*******************
            _AxoWriteBoolParameter_ParameterNumber  := AxoWriteBoolParameter_ParameterNumber;
            _AxoWriteBoolParameter_Value            := AxoWriteBoolParameter_Value;
            _AxoWriteBoolParameter_ExecutionMode    := AxoWriteBoolParameter_ExecutionMode;
            //***********ReadDigitalInput*********************
            _AxoReadDigitalInput_InputNumber        := AxoReadDigitalInput_InputNumber;
            //***********ReadDigitalOutput********************
            _AxoReadDigitalOutput_OutputNumber      := AxoReadDigitalOutput_OutputNumber;
            //***********WriteDigitalOutput*******************
            _AxoWriteDigitalOutput_OutputNumber     := AxoWriteDigitalOutput_OutputNumber;
            _AxoWriteDigitalOutput_Value            := AxoWriteDigitalOutput_Value;
            _AxoWriteDigitalOutput_ExecutionMode    := AxoWriteDigitalOutput_ExecutionMode;
            //***********ReadMotionState**********************
            _AxoReadMotionState_Source              := AxoReadMotionState_Source;
            //***********Jog**********************************
            _AxoJog_Velocity                        := AxoJog_Velocity;
            _AxoJog_Acceleration                    := AxoJog_Acceleration;
            _AxoJog_Deceleration                    := AxoJog_Deceleration;
            _AxoJog_Jerk                            := AxoJog_Jerk;
            _AxoJog_Direction                       := AxoJog_Direction;
            _AxoJogInVelocity                       := AxoJogInVelocity;
            _AxoJog_Active                          := AxoJog_Active;
        END_METHOD
